TYPE "TAx_Alarms"
VERSION : 0.1
// Block: TAx_Alarms
   STRUCT
      TOAxis : Bool;
      MCFunction : Bool;
      Drive : Bool;
      LimitMinus : Bool;
      LimitPlus : Bool;
   END_STRUCT;

END_TYPE
